FUNCTION_BLOCK CruiseController_HCECC (* Basic HCECC Function Block Type *)
  (* Standard: 61499-2 *)
  (* Version 0.0, 2007-06-26, GDS, University of Auckland *)
  (* Compiler header: package fb.rt.benchmarks.cruisecontrol; *)
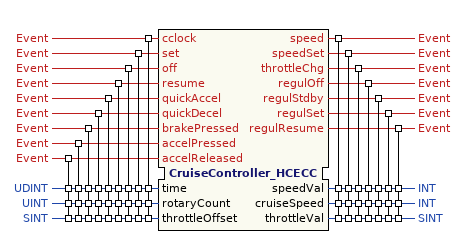
  EVENT_INPUT
    cclock WITH time, rotaryCount, throttleOffset;
    set WITH time, rotaryCount, throttleOffset;
    off WITH time, rotaryCount, throttleOffset;
    resume WITH time, rotaryCount, throttleOffset;
    quickAccel WITH time, rotaryCount, throttleOffset;
    quickDecel WITH time, rotaryCount, throttleOffset;
    brakePressed WITH time, rotaryCount, throttleOffset;
    accelPressed WITH time, rotaryCount, throttleOffset;
    accelReleased WITH time, rotaryCount, throttleOffset;
  END_EVENT
  EVENT_OUTPUT
    speed WITH speedVal, cruiseSpeed, throttleVal;
    speedSet WITH speedVal, cruiseSpeed, throttleVal;
    throttleChg WITH speedVal, cruiseSpeed, throttleVal;
    regulOff WITH speedVal, cruiseSpeed, throttleVal;
    regulStdby WITH speedVal, cruiseSpeed, throttleVal;
    regulSet WITH speedVal, cruiseSpeed, throttleVal;
    regulResume WITH speedVal, cruiseSpeed, throttleVal;
  END_EVENT
  VAR_INPUT
    time : UDINT; (* 10ms tick *)
    rotaryCount : UINT;
    throttleOffset : SINT;
  END_VAR
  VAR_OUTPUT
    speedVal : INT; (* Output event qualifier *)
    cruiseSpeed : INT;
    throttleVal : SINT;
  END_VAR
  VAR
    cruiseOn : BOOL; (* Instead of event between Manager and Throttle *)
    prevOffset : SINT := 0; (* From throttle *)
    tmp : SINT := 0; (* From throttle *)
    prevCount : UINT := 0; (* From SpeedGauge *)
    prevTime : UDINT := 0; (* From SpeedGauge *)
    count : USINT; (* From SpeedGauge *)
    desiredSpeed : INT := 0; (* From Manager *)
  END_VAR
  ALGORITHM calcSpeed IN ST:
IF rotaryCount >= prevCount THEN
    count := rotaryCount - prevCount;
ELSE
    count := 1000 + rotaryCount - prevCount;
END_IF;

IF speedVal = 0 THEN
    speedVal := (count * 7012) / 10000;
ELSE
    speedVal := (count * 7012) / 10000;
END_IF;

prevTime := time;
prevCount := rotaryCount;
  END_ALGORITHM
  ALGORITHM off IN ST:
desiredSpeed := 0;
cruiseSpeed := 0;
cruiseOn := FALSE;
  END_ALGORITHM
  ALGORITHM set IN ST:
desiredSpeed := speedVal;
cruiseSpeed := desiredSpeed;
cruiseOn := TRUE;
  END_ALGORITHM
  ALGORITHM resume IN ST:
cruiseSpeed := desiredSpeed;
cruiseOn := TRUE;
  END_ALGORITHM
  ALGORITHM standby IN ST:
cruiseSpeed := 0;
cruiseOn := FALSE;
  END_ALGORITHM
  ALGORITHM accel IN ST:
IF desiredSpeed < 165 THEN
    desiredSpeed := desiredSpeed + 5;
    cruiseSpeed := desiredSpeed;
END_IF;
  END_ALGORITHM
  ALGORITHM decel IN ST:
IF desiredSpeed >= 5 THEN
    desiredSpeed := desiredSpeed - 5;
    cruiseSpeed := desiredSpeed;
ELSE desiredSpeed := 0;
 END_IF;
  END_ALGORITHM
  ALGORITHM normal IN ST:
throttleVal := throttleOffset;
prevOffset := 0;
  END_ALGORITHM
  ALGORITHM carAccel IN ST:
throttleVal := throttleVal + throttleOffset - prevOffset;
prevOffset := throttleOffset;
  END_ALGORITHM
  ALGORITHM cruise IN ST:
tmp := (cruiseSpeed - speedVal);
tmp := tmp * 3;
 IF tmp > 45 THEN
    tmp := 45;
ELSIF tmp < 0 THEN
    tmp := 0;
 END_IF;
 throttleVal := tmp;
  END_ALGORITHM
END_FUNCTION_BLOCK
(* other elements stored in the file *)
(* ECC Name=SpeedGauge *)
(* ECState Name=START Comment=Initial State *)
(* ECState Name=CALC *)
(* ECAction Output=speed Algorithm=calcSpeed *)
(* ECTransition Destination=CALC Source=START Condition=cclock *)
(* ECTransition Destination=CALC Source=CALC Condition=cclock *)
(* ECC Name=CruiseManager *)
(* ECState Name=OFF Comment=Initial State *)
(* ECAction Output=regulOff Algorithm=off *)
(* ECState Name=SET *)
(* ECAction Output=regulSet Algorithm=set *)
(* ECState Name=STDBY *)
(* ECAction Output=regulStdby Algorithm=standby *)
(* ECState Name=RESUME *)
(* ECAction Output=regulResume Algorithm=resume *)
(* ECState Name=ACCEL *)
(* ECAction Output=speedSet Algorithm=accel *)
(* ECState Name=DECEL *)
(* ECAction Output=speedSet Algorithm=decel *)
(* ECTransition Destination=SET Source=OFF Condition=set&speedVal>50&speedVal<170 *)
(* ECTransition Destination=OFF Source=SET Condition=off *)
(* ECTransition Destination=SET Source=SET Condition=set&speedVal>50&speedVal<170 *)
(* ECTransition Destination=STDBY Source=SET Condition=brakePressed *)
(* ECTransition Destination=ACCEL Source=SET Condition=quickAccel *)
(* ECTransition Destination=DECEL Source=SET Condition=quickDecel *)
(* ECTransition Destination=OFF Source=STDBY Condition=off *)
(* ECTransition Destination=SET Source=STDBY Condition=set&speedVal>50&speedVal<170 *)
(* ECTransition Destination=RESUME Source=STDBY Condition=resume *)
(* ECTransition Destination=OFF Source=RESUME Condition=off *)
(* ECTransition Destination=SET Source=RESUME Condition=set&speedVal>50&speedVal<170 *)
(* ECTransition Destination=STDBY Source=RESUME Condition=brakePressed *)
(* ECTransition Destination=ACCEL Source=RESUME Condition=quickAccel *)
(* ECTransition Destination=DECEL Source=RESUME Condition=quickDecel *)
(* ECTransition Destination=OFF Source=ACCEL Condition=off *)
(* ECTransition Destination=SET Source=ACCEL Condition=set&speedVal>50&speedVal<170 *)
(* ECTransition Destination=STDBY Source=ACCEL Condition=brakePressed *)
(* ECTransition Destination=ACCEL Source=ACCEL Condition=quickAccel *)
(* ECTransition Destination=DECEL Source=ACCEL Condition=quickDecel *)
(* ECTransition Destination=OFF Source=DECEL Condition=off *)
(* ECTransition Destination=SET Source=DECEL Condition=set&speedVal>50&speedVal<170 *)
(* ECTransition Destination=STDBY Source=DECEL Condition=brakePressed *)
(* ECTransition Destination=ACCEL Source=DECEL Condition=quickAccel *)
(* ECTransition Destination=DECEL Source=DECEL Condition=quickDecel *)
(* ECC Name=Throttle *)
(* ECState Name=NORMAL *)
(* ECAction Output=throttleChg Algorithm=normal *)
(* ECState Name=CRUISE *)
(* ECAction Output=throttleChg Algorithm=cruise *)
(* ECState Name=ACCEL *)
(* ECAction Output=throttleChg Algorithm=carAccel *)
(* ECTransition Destination=CRUISE Source=NORMAL Condition=cruiseOn *)
(* ECTransition Destination=NORMAL Source=NORMAL Condition=accelPressed *)
(* ECTransition Destination=NORMAL Source=NORMAL Condition=accelReleased *)
(* ECTransition Destination=NORMAL Source=NORMAL Condition=cclock *)
(* ECTransition Destination=NORMAL Source=CRUISE Condition=!cruiseOn *)
(* ECTransition Destination=ACCEL Source=CRUISE Condition=accelPressed *)
(* ECTransition Destination=CRUISE Source=CRUISE Condition=cruiseOn *)
(* ECTransition Destination=CRUISE Source=CRUISE Condition=quickAccel *)
(* ECTransition Destination=CRUISE Source=CRUISE Condition=quickDecel *)
(* ECTransition Destination=CRUISE Source=CRUISE Condition=cclock *)
(* ECTransition Destination=NORMAL Source=ACCEL Condition=!cruiseOn *)
(* ECTransition Destination=CRUISE Source=ACCEL Condition=accelReleased *)
(* ECTransition Destination=ACCEL Source=ACCEL Condition=cclock *)
